FUNCTION_BLOCK MACHADO_SFC_VIEW (* Composite Function Block Type *)
  (* Standard: 61499-2 *)
  (* Version 0.2, 2003-12-05, JHC, Rockwell Automation, Renamed from NEWCOMPFB. *)
  (* Version 0.1, 2002-01-08, JHC, Rockwell Automation, Added DLY FB as example. *)
  (* Version 0.0, 2000-05-27, JHC, Rockwell Automation *)
  (* Compiler header: package fb.rt.pnp;import fb.rt.vhmi.*; *)
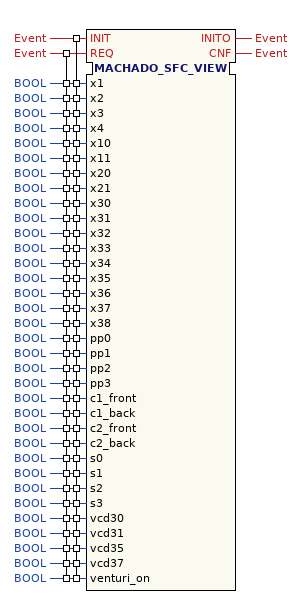
  EVENT_INPUT
    INIT WITH x1, x2, x3, x4, pp1, pp2, pp3, x10, x11, x20, x21, c1_front, c1_back, c2_front, c2_back, s1, s3, x30, x31, x32, s2, x33, x34, x35, x36, x37, x38, vcd30, venturi_on, s0, pp0, vcd31, vcd35, vcd37; (* Initialization Request *)
    REQ WITH x1, x2, x3, x4, pp1, pp2, pp3, c1_front, c1_back, c2_front, c2_back, x10, x11, x20, x21, s1, s3, x30, x31, x32, s2, x33, x34, x35, x36, x37, x38, vcd30, venturi_on, s0, pp0, vcd31, vcd35, vcd37; (* Normal Execution Request *)
  END_EVENT
  EVENT_OUTPUT
    INITO; (* Initialization Confirm *)
    CNF;
  END_EVENT
  VAR_INPUT
    x1 : BOOL; (* Input event qualifier *)
    x2 : BOOL;
    x3 : BOOL;
    x4 : BOOL;
    x10 : BOOL;
    x11 : BOOL;
    x20 : BOOL;
    x21 : BOOL;
    x30 : BOOL;
    x31 : BOOL;
    x32 : BOOL;
    x33 : BOOL;
    x34 : BOOL;
    x35 : BOOL;
    x36 : BOOL;
    x37 : BOOL;
    x38 : BOOL;
    pp0 : BOOL;
    pp1 : BOOL;
    pp2 : BOOL;
    pp3 : BOOL;
    c1_front : BOOL;
    c1_back : BOOL;
    c2_front : BOOL;
    c2_back : BOOL;
    s0 : BOOL;
    s1 : BOOL;
    s2 : BOOL;
    s3 : BOOL;
    vcd30 : BOOL;
    vcd31 : BOOL;
    vcd35 : BOOL;
    vcd37 : BOOL;
    venturi_on : BOOL;
  END_VAR
  FBS
    COORD : SFC_COORD;
    SFC2_SFC3 : SFC2_SFC3_VIEW;
    SFC1_VIEW : SFC1_VIEW;
    SFC4_VIEW : SFC4_VIEW;
    NotVcd31 : NotGate;
    NotVcd37 : NotGate;
  END_FBS
  EVENT_CONNECTIONS
    INIT TO COORD.INIT;
    REQ TO COORD.REQ;
    REQ TO SFC2_SFC3.REQ;
    COORD.INITO TO SFC1_VIEW.INIT;
    SFC1_VIEW.INITO TO SFC2_SFC3.INIT;
    COORD.CNF TO SFC1_VIEW.NAME_CHG;
    COORD.CNF TO SFC2_SFC3.NAME_CHG;
    REQ TO SFC1_VIEW.REQ;
    COORD.CNF TO SFC4_VIEW.NAME_CHG;
    SFC4_VIEW.INITO TO INITO;
    SFC4_VIEW.CNF TO CNF;
    NotVcd37.INITO TO NotVcd31.INIT;
    NotVcd37.CNF TO NotVcd31.REQ;
    NotVcd31.CNF TO SFC4_VIEW.REQ;
    NotVcd31.INITO TO SFC4_VIEW.INIT;
    SFC2_SFC3.INITO TO NotVcd37.INIT;
    SFC2_SFC3.CNF TO NotVcd37.REQ;
  END_CONNECTIONS
  DATA_CONNECTIONS
    x1 TO COORD.X1;
    x4 TO COORD.X4;
    c1_front TO COORD.c1front;
    c1_back TO COORD.c1back;
    c2_front TO COORD.c2front;
    c2_back TO COORD.c2back;
    x2 TO COORD.X2;
    x3 TO COORD.X3;
    COORD.X10_IMG TO SFC2_SFC3.X10_NAME;
    COORD.X11_IMG TO SFC2_SFC3.X11_NAME;
    COORD.L1C_IMG TO SFC2_SFC3.L1CGO_NAME;
    COORD.X20_IMG TO SFC2_SFC3.X20_NAME;
    COORD.X21_IMG TO SFC2_SFC3.X21_NAME;
    COORD.L2C_IMG TO SFC2_SFC3.L2CGO_NAME;
    x10 TO COORD.X10;
    x11 TO COORD.X11;
    x20 TO COORD.X20;
    x21 TO COORD.X21;
    x1 TO SFC2_SFC3.x1;
    x3 TO SFC2_SFC3.x3;
    x30 TO SFC2_SFC3.x30;
    s1 TO SFC2_SFC3.S1;
    s3 TO SFC2_SFC3.S3;
    x2 TO SFC2_SFC3.x2;
    s2 TO SFC2_SFC3.S2;
    COORD.X4_IMG TO SFC1_VIEW.x4;
    COORD.X1_IMG TO SFC1_VIEW.x1;
    COORD.X2_IMG TO SFC1_VIEW.x2;
    COORD.X3_IMG TO SFC1_VIEW.x3;
    pp1 TO SFC1_VIEW.PP1;
    pp2 TO SFC1_VIEW.PP2;
    pp3 TO SFC1_VIEW.PP3;
    COORD.X30_IMG TO SFC4_VIEW.X30_NAME;
    COORD.X31_IMG TO SFC4_VIEW.X31_NAME;
    COORD.X32_IMG TO SFC4_VIEW.X32_NAME;
    COORD.X33_IMG TO SFC4_VIEW.X33_NAME;
    COORD.X34_IMG TO SFC4_VIEW.X34_NAME;
    COORD.X35_IMG TO SFC4_VIEW.X35_NAME;
    COORD.X36_IMG TO SFC4_VIEW.X36_NAME;
    COORD.X37_IMG TO SFC4_VIEW.X37_NAME;
    COORD.X38_IMG TO SFC4_VIEW.X38_NAME;
    COORD.venturi_IMG TO SFC4_VIEW.VENTURI_NAME;
    x30 TO COORD.X30;
    x31 TO COORD.X31;
    x32 TO COORD.X32;
    x33 TO COORD.X33;
    x34 TO COORD.X34;
    x35 TO COORD.X35;
    x36 TO COORD.X36;
    x37 TO COORD.X37;
    x38 TO COORD.X38;
    venturi_on TO COORD.venturi_on;
    s0 TO SFC4_VIEW.s0;
    s1 TO SFC4_VIEW.s1;
    s2 TO SFC4_VIEW.s2;
    s3 TO SFC4_VIEW.s3;
    x1 TO SFC4_VIEW.x1;
    x2 TO SFC4_VIEW.x2;
    x3 TO SFC4_VIEW.x3;
    venturi_on TO SFC4_VIEW.vacuum;
    x11 TO SFC4_VIEW.x11;
    x21 TO SFC4_VIEW.x21;
    pp0 TO SFC4_VIEW.pp0;
    COORD.L1CGI_IMG TO SFC4_VIEW.L1CGI_NAME;
    COORD.L2CGI_IMG TO SFC4_VIEW.L2CGI_NAME;
    vcd30 TO COORD.vcd30;
    vcd31 TO COORD.vcd31;
    vcd35 TO COORD.vcd35;
    vcd37 TO COORD.vcd37;
    COORD.vcd30_IMG TO SFC4_VIEW.VCGD30_NAME;
    COORD.vcd31_IMG TO SFC4_VIEW.VCGD31_NAME;
    COORD.vcd35_IMG TO SFC4_VIEW.VCGD35_NAME;
    COORD.vcd37_IMG TO SFC4_VIEW.VCGD37_NAME;
    vcd30 TO SFC4_VIEW.vcd30;
    vcd35 TO SFC4_VIEW.vcd35;
    NotVcd31.QO TO SFC4_VIEW.vcu31;
    NotVcd37.QO TO SFC4_VIEW.vcu37;
    vcd31 TO NotVcd31.QI;
    vcd37 TO NotVcd37.QI;
  END_CONNECTIONS
END_FUNCTION_BLOCK
